      Especial_M460 : Bool;
      Bit_02_M460 : Bool;
      Retroceder_M460 : Bool;
      Retirar_M460 : Bool;
      Continuar_M460 : Bool;
      Entrar_M460 : Bool;
      EmiOK_M460 : Bool;
      FinLote_M461 : Bool;
      Especial_M461 : Bool;
      Bit_02_M461 : Bool;
      Retroceder_M461 : Bool;
      Retirar_M461 : Bool;
      Continuar_M461 : Bool;
      Entrar_M461 : Bool;
      EmiOK_M461 : Bool;
      FinLote_M462 : Bool;
      Especial_M462 : Bool;
      Bit_02_M462 : Bool;
      Retroceder_M462 : Bool;
      Retirar_M462 : Bool;
      Continuar_M462 : Bool;
      Entrar_M462 : Bool;
      EmiOK_M462 : Bool;
      FinLote_M463 : Bool;
      Especial_M463 : Bool;
      Bit_02_M463 : Bool;
      Retroceder_M463 : Bool;
      Retirar_M463 : Bool;
      Continuar_M463 : Bool;
      Entrar_M463 : Bool;
      EmiOK_M463 : Bool;
      FinLote_M464 : Bool;
      Especial_M464 : Bool;
      Bit_02_M464 : Bool;
      Retroceder_M464 : Bool;
      Retirar_M464 : Bool;
      Continuar_M464 : Bool;
      Entrar_M464 : Bool;
      EmiOK_M464 : Bool;
      FinLote_M465 : Bool;
      Especial_M465 : Bool;
      Bit_02_M465 : Bool;
      Retroceder_M465 : Bool;
      Retirar_M465 : Bool;
      Continuar_M465 : Bool;
      Entrar_M465 : Bool;
      EmiOK_M465 : Bool;
      FinLote_M466 : Bool;
      Especial_M466 : Bool;
      Bit_02_M466 : Bool;
      Retroceder_M466 : Bool;
      Retirar_M466 : Bool;
      Continuar_M466 : Bool;
      Entrar_M466 : Bool;
      EmiOK_M466 : Bool;
      FinLote_M467 : Bool;
      Especial_M467 : Bool;
      Bit_02_M467 : Bool;
      Retroceder_M467 : Bool;
      Retirar_M467 : Bool;
      Continuar_M467 : Bool;
      Entrar_M467 : Bool;
      EmiOK_M467 : Bool;
      FinLote_M468 : Bool;
      Especial_M468 : Bool;
      Bit_02_M468 : Bool;
      Retroceder_M468 : Bool;
      Retirar_M468 : Bool;
      Continuar_M468 : Bool;
      Entrar_M468 : Bool;
      EmiOK_M468 : Bool;
      FinLote_M469 : Bool;
      Especial_M469 : Bool;
      Bit_02_M469 : Bool;
      Retroceder_M469 : Bool;
      Retirar_M469 : Bool;
      Continuar_M469 : Bool;
      Entrar_M469 : Bool;
      EmiOK_M469 : Bool;
      FinLote_M470 : Bool;
      Especial_M470 : Bool;
      Bit_02_M470 : Bool;
      Retroceder_M470 : Bool;
      Retirar_M470 : Bool;
      Continuar_M470 : Bool;
      Entrar_M470 : Bool;
      EmiOK_M470 : Bool;
      FinLote_M471 : Bool;
      Especial_M471 : Bool;
      Bit_02_M471 : Bool;
      Retroceder_M471 : Bool;
      Retirar_M471 : Bool;
      Continuar_M471 : Bool;
      Entrar_M471 : Bool;
      EmiOK_M471 : Bool;
      FinLote_M472 : Bool;
      Especial_M472 : Bool;
      Bit_02_M472 : Bool;
      Retroceder_M472 : Bool;
      Retirar_M472 : Bool;
      Continuar_M472 : Bool;
      Entrar_M472 : Bool;
      EmiOK_M472 : Bool;
      FinLote_M473 : Bool;
      Especial_M473 : Bool;
      Bit_02_M473 : Bool;
      Retroceder_M473 : Bool;
      Retirar_M473 : Bool;
      Continuar_M473 : Bool;
      Entrar_M473 : Bool;
      EmiOK_M473 : Bool;
      FinLote_M474 : Bool;
      Especial_M474 : Bool;
      Bit_02_M474 : Bool;
      Retroceder_M474 : Bool;
      Retirar_M474 : Bool;
      Continuar_M474 : Bool;
      Entrar_M474 : Bool;
      EmiOK_M474 : Bool;
      FinLote_M475 : Bool;
      Especial_M475 : Bool;
      Bit_02_M475 : Bool;
      Retroceder_M475 : Bool;
      Retirar_M475 : Bool;
      Continuar_M475 : Bool;
      Entrar_M475 : Bool;
      EmiOK_M475 : Bool;
      FinLote_M476 : Bool;
      Especial_M476 : Bool;
      Bit_02_M476 : Bool;
      Retroceder_M476 : Bool;
      Retirar_M476 : Bool;
      Continuar_M476 : Bool;
      Entrar_M476 : Bool;
      EmiOK_M476 : Bool;
      FinLote_M477 : Bool;
      Especial_M477 : Bool;
      Bit_02_M477 : Bool;
      Retroceder_M477 : Bool;
      Retirar_M477 : Bool;
      Continuar_M477 : Bool;
      Entrar_M477 : Bool;
      EmiOK_M477 : Bool;
      FinLote_M478 : Bool;
      Especial_M478 : Bool;
      Bit_02_M478 : Bool;
      Retroceder_M478 : Bool;
      Retirar_M478 : Bool;
      Continuar_M478 : Bool;
      Entrar_M478 : Bool;
      EmiOK_M478 : Bool;
      FinLote_M479 : Bool;
      Especial_M479 : Bool;
      Bit_02_M479 : Bool;
      Retroceder_M479 : Bool;
      Retirar_M479 : Bool;
      Continuar_M479 : Bool;
      Entrar_M479 : Bool;
      EmiOK_M479 : Bool;
      FinLote_M480 : Bool;
      Especial_M480 : Bool;
      Bit_02_M480 : Bool;
      Retroceder_M480 : Bool;
      Retirar_M480 : Bool;
      Continuar_M480 : Bool;
      Entrar_M480 : Bool;
      EmiOK_M480 : Bool;
      FinLote_M481 : Bool;
      Especial_M481 : Bool;
      Bit_02_M481 : Bool;
      Retroceder_M481 : Bool;
      Retirar_M481 : Bool;
      Continuar_M481 : Bool;
      Entrar_M481 : Bool;
      EmiOK_M481 : Bool;
      FinLote_M482 : Bool;
      Especial_M482 : Bool;
      Bit_02_M482 : Bool;
      Retroceder_M482 : Bool;
      Retirar_M482 : Bool;
      Continuar_M482 : Bool;
      Entrar_M482 : Bool;
      EmiOK_M482 : Bool;
      FinLote_M483 : Bool;
      Especial_M483 : Bool;
      Bit_02_M483 : Bool;
      Retroceder_M483 : Bool;
      Retirar_M483 : Bool;
      Continuar_M483 : Bool;
      Entrar_M483 : Bool;
      EmiOK_M483 : Bool;
      FinLote_M484 : Bool;
      Especial_M484 : Bool;
      Bit_02_M484 : Bool;
      Retroceder_M484 : Bool;
      Retirar_M484 : Bool;
      Continuar_M484 : Bool;
      Entrar_M484 : Bool;
      EmiOK_M484 : Bool;
      FinLote_M485 : Bool;
      Especial_M485 : Bool;
      Bit_02_M485 : Bool;
      Retroceder_M485 : Bool;
      Retirar_M485 : Bool;
      Continuar_M485 : Bool;
      Entrar_M485 : Bool;
      EmiOK_M485 : Bool;
      FinLote_M486 : Bool;
      Especial_M486 : Bool;
      Bit_02_M486 : Bool;
      Retroceder_M486 : Bool;
      Retirar_M486 : Bool;
      Continuar_M486 : Bool;
      Entrar_M486 : Bool;
      EmiOK_M486 : Bool;
      FinLote_M487 : Bool;
      Especial_M487 : Bool;
      Bit_02_M487 : Bool;
      Retroceder_M487 : Bool;
      Retirar_M487 : Bool;
      Continuar_M487 : Bool;
      Entrar_M487 : Bool;
      EmiOK_M487 : Bool;
      FinLote_M488 : Bool;
      Especial_M488 : Bool;
      Bit_02_M488 : Bool;
      Retroceder_M488 : Bool;
      Retirar_M488 : Bool;
      Continuar_M488 : Bool;
      Entrar_M488 : Bool;
      EmiOK_M488 : Bool;
      FinLote_M489 : Bool;
      Especial_M489 : Bool;
      Bit_02_M489 : Bool;
      Retroceder_M489 : Bool;
      Retirar_M489 : Bool;
      Continuar_M489 : Bool;
      Entrar_M489 : Bool;
      EmiOK_M489 : Bool;
      FinLote_M490 : Bool;
      Especial_M490 : Bool;
      Bit_02_M490 : Bool;
      Retroceder_M490 : Bool;
      Retirar_M490 : Bool;
      Continuar_M490 : Bool;
      Entrar_M490 : Bool;
      EmiOK_M490 : Bool;
      FinLote_M491 : Bool;
      Especial_M491 : Bool;
      Bit_02_M491 : Bool;
      Retroceder_M491 : Bool;
      Retirar_M491 : Bool;
      Continuar_M491 : Bool;
      Entrar_M491 : Bool;
      EmiOK_M491 : Bool;
      FinLote_M492 : Bool;
      Especial_M492 : Bool;
      Bit_02_M492 : Bool;
      Retroceder_M492 : Bool;
      Retirar_M492 : Bool;
      Continuar_M492 : Bool;
      Entrar_M492 : Bool;
      EmiOK_M492 : Bool;
      FinLote_M493 : Bool;
      Especial_M493 : Bool;
      Bit_02_M493 : Bool;
      Retroceder_M493 : Bool;
      Retirar_M493 : Bool;
      Continuar_M493 : Bool;
      Entrar_M493 : Bool;
      EmiOK_M493 : Bool;
      FinLote_M494 : Bool;
      Especial_M494 : Bool;
      Bit_02_M494 : Bool;
      Retroceder_M494 : Bool;
      Retirar_M494 : Bool;
      Continuar_M494 : Bool;
      Entrar_M494 : Bool;
      EmiOK_M494 : Bool;
      FinLote_M495 : Bool;
      Especial_M495 : Bool;
      Bit_02_M495 : Bool;
      Retroceder_M495 : Bool;
      Retirar_M495 : Bool;
      Continuar_M495 : Bool;
      Entrar_M495 : Bool;
      EmiOK_M495 : Bool;
      FinLote_M496 : Bool;
      Especial_M496 : Bool;
      Bit_02_M496 : Bool;
      Retroceder_M496 : Bool;
      Retirar_M496 : Bool;
      Continuar_M496 : Bool;
      Entrar_M496 : Bool;
      EmiOK_M496 : Bool;
      FinLote_M497 : Bool;
      Especial_M497 : Bool;
      Bit_02_M497 : Bool;
      Retroceder_M497 : Bool;
      Retirar_M497 : Bool;
      Continuar_M497 : Bool;
      Entrar_M497 : Bool;
      EmiOK_M497 : Bool;
      FinLote_M498 : Bool;
      Especial_M498 : Bool;
      Bit_02_M498 : Bool;
      Retroceder_M498 : Bool;
      Retirar_M498 : Bool;
      Continuar_M498 : Bool;
      Entrar_M498 : Bool;
      EmiOK_M498 : Bool;
      FinLote_M499 : Bool;
      Especial_M499 : Bool;
      Bit_02_M499 : Bool;
      Retroceder_M499 : Bool;
      Retirar_M499 : Bool;
      Continuar_M499 : Bool;
      Entrar_M499 : Bool;
      EmiOK_M499 : Bool;
      FinLote_M500 : Bool;
      Especial_M500 : Bool;
      Bit_02_M500 : Bool;
      Retroceder_M500 : Bool;
      Retirar_M500 : Bool;
      Continuar_M500 : Bool;
      Entrar_M500 : Bool;
      EmiOK_M500 : Bool;
      Bit_00_CCPIF : Bool;
      Bit_01_CCPIF : Bool;
      Rearme_CCPIF : Bool;
      Bit_03_CCPIF : Bool;
      Reset_CCPIF : Bool;
      Paro_CCPIF : Bool;
      Marcha_CCPIF : Bool;
      EmiOK_CCPIF : Bool;
      Bit_00_CBOX1 : Bool;
      Bit_01_CBOX1 : Bool;
      Rearme_CBOX1 : Bool;
      Bit_03_CBOX1 : Bool;
      Reset_CBOX1 : Bool;
      Paro_CBOX1 : Bool;
      Marcha_CBOX1 : Bool;
      EmiOK_CBOX1 : Bool;
      Bit_00_CBOX2 : Bool;
      Bit_01_CBOX2 : Bool;
      Rearme_CBOX2 : Bool;
      Bit_03_CBOX2 : Bool;
      Reset_CBOX2 : Bool;
      Paro_CBOX2 : Bool;
      Marcha_CBOX2 : Bool;
      EmiOK_CBOX2 : Bool;
      Bit_00_CBOX3 : Bool;
      Bit_01_CBOX3 : Bool;
      Rearme_CBOX3 : Bool;
      Bit_03_CBOX3 : Bool;
      Reset_CBOX3 : Bool;
      Paro_CBOX3 : Bool;
      Marcha_CBOX3 : Bool;
      EmiOK_CBOX3 : Bool;
      Bit_00_CBOX4 : Bool;
      Bit_01_CBOX4 : Bool;
      Rearme_CBOX4 : Bool;
      Bit_03_CBOX4 : Bool;
      Reset_CBOX4 : Bool;
      Paro_CBOX4 : Bool;
      Marcha_CBOX4 : Bool;
      EmiOK_CBOX4 : Bool;
      Bit_00_CBOX5 : Bool;
      Bit_01_CBOX5 : Bool;
      Rearme_CBOX5 : Bool;
      Bit_03_CBOX5 : Bool;
      Reset_CBOX5 : Bool;
      Paro_CBOX5 : Bool;
      Marcha_CBOX5 : Bool;
      EmiOK_CBOX5 : Bool;
      Bit_00_CBOX6 : Bool;
      Bit_01_CBOX6 : Bool;
      Rearme_CBOX6 : Bool;
      Bit_03_CBOX6 : Bool;
      Reset_CBOX6 : Bool;
      Paro_CBOX6 : Bool;
      Marcha_CBOX6 : Bool;
      EmiOK_CBOX6 : Bool;
      Bit_00_CBOX7 : Bool;
      Bit_01_CBOX7 : Bool;
      Rearme_CBOX7 : Bool;
      Bit_03_CBOX7 : Bool;
      Reset_CBOX7 : Bool;
      Paro_CBOX7 : Bool;
      Marcha_CBOX7 : Bool;
      EmiOK_CBOX7 : Bool;
      Bit_00_CBOX8 : Bool;
      Bit_01_CBOX8 : Bool;
      Rearme_CBOX8 : Bool;
      Bit_03_CBOX8 : Bool;
      Reset_CBOX8 : Bool;
      Paro_CBOX8 : Bool;
      Marcha_CBOX8 : Bool;
      EmiOK_CBOX8 : Bool;
      Bit_00_CBOX9 : Bool;
      Bit_01_CBOX9 : Bool;
      Rearme_CBOX9 : Bool;
      Bit_03_CBOX9 : Bool;
      Reset_CBOX9 : Bool;
      Paro_CBOX9 : Bool;
      Marcha_CBOX9 : Bool;
      EmiOK_CBOX9 : Bool;
      Especial : Array[1..128] of Word;
   END_VAR
BEGIN
END_DATA_BLOCK
